FUNCTION_BLOCK FeedPumpFbReactor (* Basic Function Block Type *)
  (* Standard: 61499-2 *)
  (* Version 0.0, 7/13/2026, Schneider Electric, Template *)
  PACKAGE SE.Nereda;
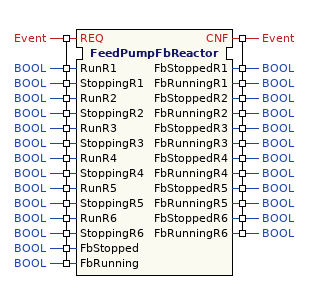
  EVENT_INPUT
    REQ WITH RunR1, RunR2, RunR3, RunR4, RunR5, RunR6, StoppingR1, StoppingR2, StoppingR3, StoppingR4, StoppingR5, StoppingR6, FbStopped, FbRunning; (* Normal Execution Request *)
  END_EVENT
  EVENT_OUTPUT
    CNF WITH FbStoppedR1, FbStoppedR2, FbStoppedR3, FbStoppedR4, FbStoppedR5, FbStoppedR6, FbRunningR1, FbRunningR2, FbRunningR3, FbRunningR4, FbRunningR5, FbRunningR6; (* Execution Confirmation *)
  END_EVENT
  VAR_INPUT
    RunR1 : BOOL;
    StoppingR1 : BOOL;
    RunR2 : BOOL;
    StoppingR2 : BOOL;
    RunR3 : BOOL;
    StoppingR3 : BOOL;
    RunR4 : BOOL;
    StoppingR4 : BOOL;
    RunR5 : BOOL;
    StoppingR5 : BOOL;
    RunR6 : BOOL;
    StoppingR6 : BOOL;
    FbStopped : BOOL;
    FbRunning : BOOL;
  END_VAR
  VAR_OUTPUT
    FbStoppedR1 : BOOL;
    FbRunningR1 : BOOL;
    FbStoppedR2 : BOOL;
    FbRunningR2 : BOOL;
    FbStoppedR3 : BOOL;
    FbRunningR3 : BOOL;
    FbStoppedR4 : BOOL;
    FbRunningR4 : BOOL;
    FbStoppedR5 : BOOL;
    FbRunningR5 : BOOL;
    FbStoppedR6 : BOOL;
    FbRunningR6 : BOOL;
  END_VAR
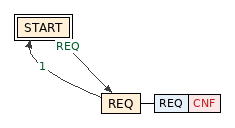
  EC_STATES
    START; (* Initial State *)
    REQ : REQ -> CNF;
  END_STATES
  EC_TRANSITIONS
    START TO REQ := REQ;
    REQ TO START := 1;
  END_TRANSITIONS
  ALGORITHM INIT IN ST: (* Initialization algorithm *)
;
  END_ALGORITHM
  ALGORITHM REQ IN ST: (* Normally executed algorithm *)
;
IF NOT RunR1 AND NOT RunR2 AND NOT RunR3 AND NOT RunR4 AND NOT RunR5 AND NOT RunR6 THEN
	FbRunningR1 := FbRunning;
	FbStoppedR1 := FbStopped;

	FbRunningR2 := FbRunning;
	FbStoppedR2 := FbStopped;

	FbRunningR3 := FbRunning;
	FbStoppedR3 := FbStopped;

	FbRunningR4 := FbRunning;
	FbStoppedR4 := FbStopped;

	FbRunningR5 := FbRunning;
	FbStoppedR5 := FbStopped;

	FbRunningR6 := FbRunning;
	FbStoppedR6 := FbStopped;
ELSE
	IF StoppingR1 THEN
		FbRunningR1 := FALSE;
		FbStoppedR1 := TRUE;
	END_IF;

	IF StoppingR2 THEN
		FbRunningR2 := FALSE;
		FbStoppedR2 := TRUE;
	END_IF;

	IF StoppingR3 THEN
		FbRunningR3 := FALSE;
		FbStoppedR3 := TRUE;
	END_IF;

	IF StoppingR4 THEN
		FbRunningR4 := FALSE;
		FbStoppedR4 := TRUE;
	END_IF;

	IF StoppingR5 THEN
		FbRunningR5 := FALSE;
		FbStoppedR5 := TRUE;
	END_IF;

	IF StoppingR6 THEN
		FbRunningR6 := FALSE;
		FbStoppedR6 := TRUE;
	END_IF;
END_IF;
  END_ALGORITHM
END_FUNCTION_BLOCK
